(* Schneider Machine Expert - Basic project Project1_Part2, file version 1.6.0.0 *)
(* ProjectInformations: Name=New project *)

HARDWARE
  Cpu 0: TM221M16R/G
  EthernetConfiguration: NetworkName=M221, IpAllocationMode=FixedAddress, IpAddress=0.0.0.0, SubnetMask=0.0.0.0
  SerialLineConfiguration: Baud=Baud19200, Parity=ParityEven, DataBits=DataBits8, StopBits=StopBits1, PhysicalMedium=PhysicalMediumRs485, TransmissionMode=TransmissionModeModbusRtu, SlaveId=1, Addressing=SlaveAddressing
  MastTask: UsePeriodScanMode=false, PeriodScan=100
  FastTask: Period=255
  CpuBehavior: StartingMode=StartAsPreviousState, AutoSaveRamOnEeprom=true, WatchdogPeriod=250

SYMBOLS  (address, symbol, comment, settings)
  %M0       SHUTDOWN_STATE
  %M1       CHECKPOINT1
  %M2       CHECKPOINT2
  %M3       CHECKPOINT3
  %MW0      CURRENT_PRESSURE
  %KW0      PRESSURE_CHECKPOINT  [Value=500]
  %KW1      PRESSURE_CHECKPOINT_UNREACHABLE  [Value=1001]
  %TM0        [Preset=5, Base=OneSecond]
  %I0.0     SHUTDOWN
  %I0.1     CANCEL_SHUTDOWN
  %I0.2     CONFIRM_PRESSURE_CHANGE
  %I0.3     CONFIRM_SHUTDOWN
  %I0.4     EMERGENCY_SHUTDOWN
  %Q0.0     SHUTDOWN_CHECK_1
  %Q0.1     SHUTDOWN_CANCELED
  %Q0.2     SHUTDOWN_CHECK_2
  %Q0.3     SHUTDOWN_CHECK_3
  %Q0.4     EMERGENCY_SHUTDOWN_DECLARED
  %Q0.5     SHUTDOWN_COMPLETED
  %IW0.0    SET_PRESSURE  [Type=Type_0_10V, Scope=Scope_Normal, Minimum=0, Maximum=1000]

POU New POU
  (* SectionNumber=1 *)

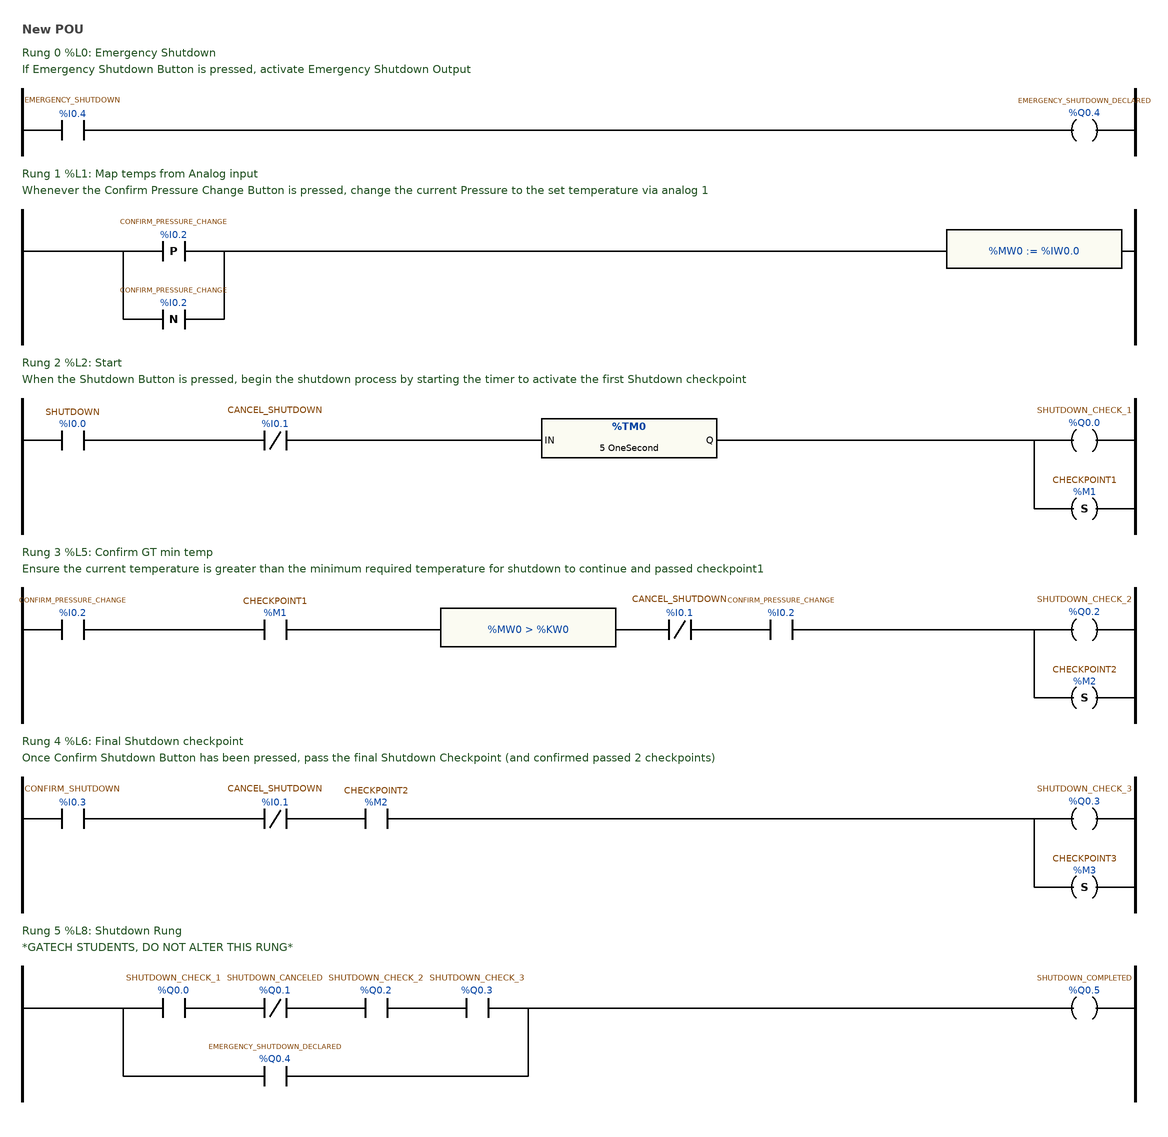

// Rung 0 %L0: Emergency Shutdown
// If Emergency Shutdown Button is pressed, activate Emergency Shutdown Output
  %L0:
  LD %I0.4                (* EMERGENCY_SHUTDOWN *)
  ST %Q0.4                (* EMERGENCY_SHUTDOWN_DECLARED *)
  // as ST:
  //   %L0:
  //   EMERGENCY_SHUTDOWN_DECLARED := EMERGENCY_SHUTDOWN;

// Rung 1 %L1: Map temps from Analog input
// Whenever the Confirm Pressure Change Button is pressed, change the current Pressure to the set temperature via analog 1
  %L1:
  LDR %I0.2               (* CONFIRM_PRESSURE_CHANGE *)
  ORF %I0.2               (* CONFIRM_PRESSURE_CHANGE *)
  [ %MW0 := %IW0.0 ]      (* CURRENT_PRESSURE, SET_PRESSURE *)
  // as ST:
  //   %L1:
  //   IF RISING(CONFIRM_PRESSURE_CHANGE) OR FALLING(CONFIRM_PRESSURE_CHANGE) THEN CURRENT_PRESSURE := SET_PRESSURE; END_IF;

// Rung 2 %L2: Start
// When the Shutdown Button is pressed, begin the shutdown process by starting the timer to activate the first Shutdown checkpoint
  %L2:
  BLK %TM0
  LD %I0.0                (* SHUTDOWN *)
  ANDN %I0.1              (* CANCEL_SHUTDOWN *)
  IN
  OUT_BLK
  LD Q
  ST %Q0.0                (* SHUTDOWN_CHECK_1 *)
  S %M1                   (* CHECKPOINT1 *)
  END_BLK
  // as ST:
  //   %L2:
  //   %TM0(IN := SHUTDOWN AND NOT CANCEL_SHUTDOWN);
  //   SHUTDOWN_CHECK_1 := %TM0.Q;
  //   IF %TM0.Q THEN CHECKPOINT1 := TRUE; END_IF;

// Rung 3 %L5: Confirm GT min temp
// Ensure the current temperature is greater than the minimum required temperature for shutdown to continue and passed checkpoint1
  %L5:
  LD %I0.2                (* CONFIRM_PRESSURE_CHANGE *)
  AND %M1                 (* CHECKPOINT1 *)
  AND [ %MW0 > %KW0 ]     (* CURRENT_PRESSURE, PRESSURE_CHECKPOINT *)
  ANDN %I0.1              (* CANCEL_SHUTDOWN *)
  AND %I0.2               (* CONFIRM_PRESSURE_CHANGE *)
  ST %Q0.2                (* SHUTDOWN_CHECK_2 *)
  S %M2                   (* CHECKPOINT2 *)
  // as ST:
  //   %L5:
  //   SHUTDOWN_CHECK_2 := CONFIRM_PRESSURE_CHANGE AND CHECKPOINT1 AND CURRENT_PRESSURE > PRESSURE_CHECKPOINT AND NOT CANCEL_SHUTDOWN AND CONFIRM_PRESSURE_CHANGE;
  //   IF CONFIRM_PRESSURE_CHANGE AND CHECKPOINT1 AND CURRENT_PRESSURE > PRESSURE_CHECKPOINT AND NOT CANCEL_SHUTDOWN AND CONFIRM_PRESSURE_CHANGE THEN CHECKPOINT2 := TRUE; END_IF;

// Rung 4 %L6: Final Shutdown checkpoint
// Once Confirm Shutdown Button has been pressed, pass the final Shutdown Checkpoint (and confirmed passed 2 checkpoints)
  %L6:
  LD %I0.3                (* CONFIRM_SHUTDOWN *)
  ANDN %I0.1              (* CANCEL_SHUTDOWN *)
  AND %M2                 (* CHECKPOINT2 *)
  ST %Q0.3                (* SHUTDOWN_CHECK_3 *)
  S %M3                   (* CHECKPOINT3 *)
  // as ST:
  //   %L6:
  //   SHUTDOWN_CHECK_3 := CONFIRM_SHUTDOWN AND NOT CANCEL_SHUTDOWN AND CHECKPOINT2;
  //   IF CONFIRM_SHUTDOWN AND NOT CANCEL_SHUTDOWN AND CHECKPOINT2 THEN CHECKPOINT3 := TRUE; END_IF;

// Rung 5 %L8: Shutdown Rung
// *GATECH STUDENTS, DO NOT ALTER THIS RUNG*
  %L8:
  LD %Q0.0                (* SHUTDOWN_CHECK_1 *)
  ANDN %Q0.1              (* SHUTDOWN_CANCELED *)
  AND %Q0.2               (* SHUTDOWN_CHECK_2 *)
  AND %Q0.3               (* SHUTDOWN_CHECK_3 *)
  OR %Q0.4                (* EMERGENCY_SHUTDOWN_DECLARED *)
  ST %Q0.5                (* SHUTDOWN_COMPLETED *)
  // as ST:
  //   %L8:
  //   SHUTDOWN_COMPLETED := SHUTDOWN_CHECK_1 AND NOT SHUTDOWN_CANCELED AND SHUTDOWN_CHECK_2 AND SHUTDOWN_CHECK_3 OR EMERGENCY_SHUTDOWN_DECLARED;

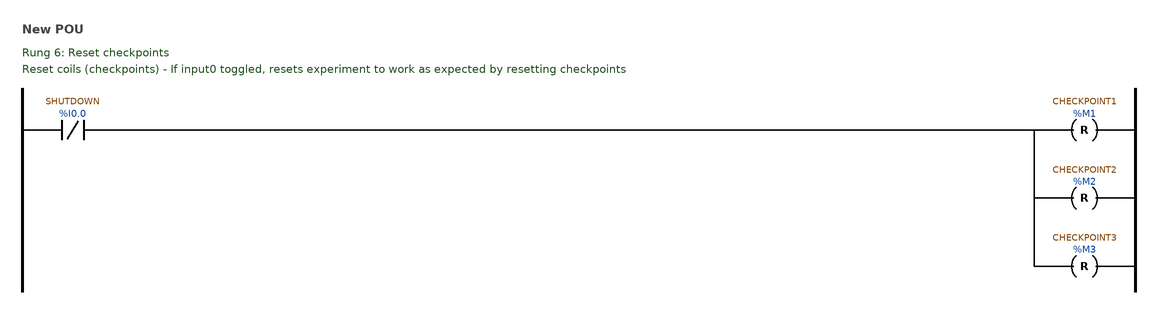

// Rung 6: Reset checkpoints
// Reset coils (checkpoints) - If input0 toggled, resets experiment to work as expected by resetting checkpoints
  LDN %I0.0               (* SHUTDOWN *)
  R %M1                   (* CHECKPOINT1 *)
  R %M2                   (* CHECKPOINT2 *)
  R %M3                   (* CHECKPOINT3 *)
  // as ST:
  //   IF NOT SHUTDOWN THEN CHECKPOINT1 := FALSE; END_IF;
  //   IF NOT SHUTDOWN THEN CHECKPOINT2 := FALSE; END_IF;
  //   IF NOT SHUTDOWN THEN CHECKPOINT3 := FALSE; END_IF;
